(* CODESYS project GVL_ROBOT.gvl.xml

Project tree, tasks and I/O mapping:
  global variables GVL_ROBOT
*)

// GVL_ROBOT
{attribute 'qualified_only'}
VAR_GLOBAL
	Command       : ST_ROBOT_COMMAND; // Выбранная команда робота
	ModbusCommand : ST_ROBOT_COMMAND; // Команда внешнему роботу
	Status        : ST_ROBOT_STATUS; // Рабочие статусы робота
	Diag          : ST_ROBOT_DIAG; // Состояние автомата робота
	Error         : ST_ROBOT_ERRORS; // Активные и последние ошибки робота

	xModbusBusy  : BOOL; // Внешний робот выполняет команду
	xModbusDone  : BOOL; // Внешний робот завершил команду
	xModbusError : BOOL; // Ошибка внешнего робота или обмена
END_VAR
